// TIA Portal V19 export
FUNCTION "MeasWheelCheckRotation_TypeExtEnc" : Int   // FC49, LAD
TITLE = Check velocity of the measuring wheel compared with velocity axis (motor)
// Da usare con encoder rotella di misura collegata come encoder esterno e che quindi non chiude l'anello di posizione di un asse
// stored: Access Published, SetENOAutomatically false
   VAR_INPUT
      TO_EncMatCounter : TO_ExternalEncoder;   // TO of the external encoder
      VelMaterialMover : LReal;   // "#TO_Ax.Velocity"of the material mover axis
      VelMin : LReal;   // Min velocity for execute check
      ErrPercentageMax : LReal;   // Max error % beetween velocity
   END_VAR
   VAR_OUTPUT
      Err : LReal;   // Show % actual error percentage
   END_VAR
   VAR_TEMP
      MeasWheelIsActive : Bool;
      MotorVelocity : LReal;
      MotorVelocityABS : LReal;
      ErrorPercentage : LReal;
      Check : Bool;
      err0 : LReal;
   END_VAR
   VAR CONSTANT
      RET_NULL : Int := 0;
      RET_VEL_OK : Int := 1;
      RET_VEL_BELOW_MIN : Int := 10;
      RET_ERR_ENC_NOT_VALID : Int := 101;
      RET_VEL_DELTA_EXCEED : Int := 103;
   END_VAR
   VAR_TEMP   // added for the SCL form of the ladder/FBD networks
      _w1 : Bool;
   END_VAR
BEGIN

REGION Network 1: Out error percentage
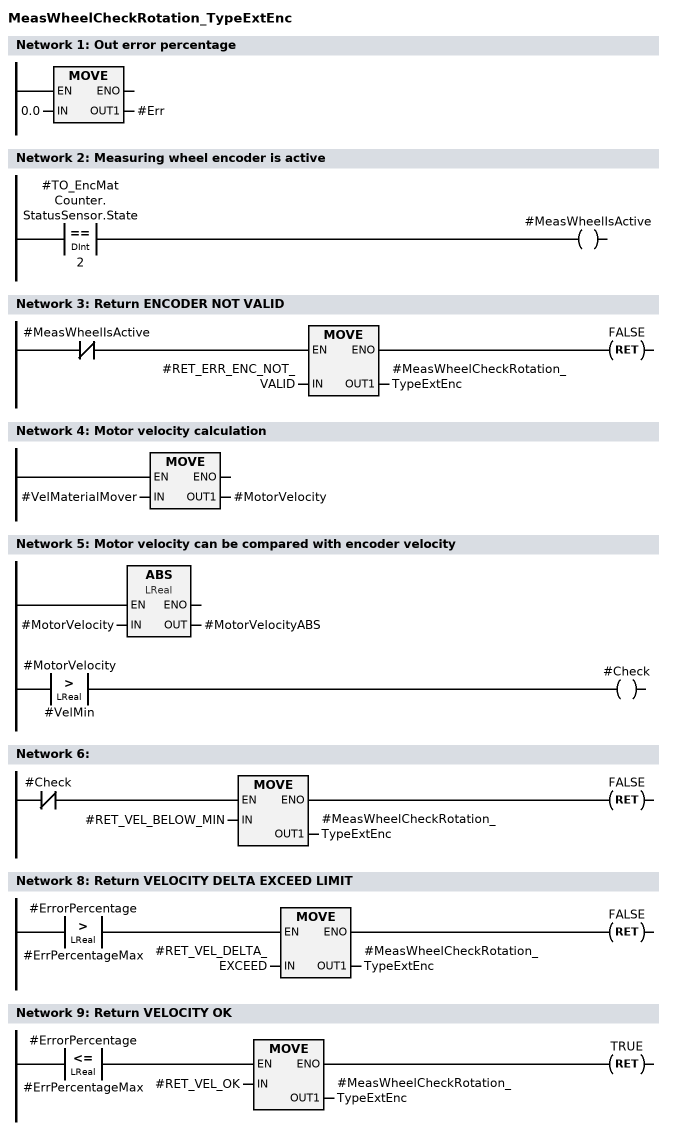
   RUNG wire#powerrail
      { S7_GenerateENO := "TRUE" } Move(in := 0.0, out1 => #Err)
   END_RUNG
   // the same network as SCL:
   #Err := 0.0;
END_REGION

REGION Network 2: Measuring wheel encoder is active
   RUNG wire#powerrail
      { S7_Templates := "SrcType := DInt" } EQ_Contact(in1 := #TO_EncMatCounter.StatusSensor.State, in2 := 2)
      Coil( #MeasWheelIsActive )
   END_RUNG
   // the same network as SCL:
   #MeasWheelIsActive := #TO_EncMatCounter.StatusSensor.State = 2;
END_REGION

REGION Network 3: Return ENCODER NOT VALID
   RUNG wire#powerrail
      I_Contact( #MeasWheelIsActive )
      { S7_GenerateENO := "TRUE" } Move(in := #RET_ERR_ENC_NOT_VALID, out1 => #MeasWheelCheckRotation_TypeExtEnc)
      ReturnCoil( FALSE )
   END_RUNG
   // the same network as SCL:
   // ENO of a box is taken as its EN; it also drops when the box reports an error
   IF NOT #MeasWheelIsActive THEN
       #MeasWheelCheckRotation_TypeExtEnc := #RET_ERR_ENC_NOT_VALID;
       ENO := FALSE;
       RETURN;
   END_IF;
END_REGION

REGION Network 4: Motor velocity calculation
   RUNG wire#powerrail
      { S7_GenerateENO := "TRUE" } Move(in := #VelMaterialMover, out1 => #MotorVelocity)
   END_RUNG
   // the same network as SCL:
   #MotorVelocity := #VelMaterialMover;
END_REGION

REGION Network 5: Motor velocity can be compared with encoder velocity
   RUNG wire#powerrail
      { S7_Templates := "SrcType := LReal"; S7_GenerateENO := "TRUE" } Abs(in := #MotorVelocity, out => #MotorVelocityABS)
   END_RUNG
   RUNG wire#powerrail
      { S7_Templates := "SrcType := LReal" } GT_Contact(in1 := #MotorVelocity, in2 := #VelMin)
      Coil( #Check )
   END_RUNG
   // the same network as SCL:
   #MotorVelocityABS := ABS(#MotorVelocity);
   #Check := #MotorVelocity > #VelMin;
END_REGION

REGION Network 6
   RUNG wire#powerrail
      I_Contact( #Check )
      { S7_GenerateENO := "TRUE" } Move(in := #RET_VEL_BELOW_MIN, out1 => #MeasWheelCheckRotation_TypeExtEnc)
      ReturnCoil( FALSE )
   END_RUNG
   // the same network as SCL:
   // ENO of a box is taken as its EN; it also drops when the box reports an error
   IF NOT #Check THEN
       #MeasWheelCheckRotation_TypeExtEnc := #RET_VEL_BELOW_MIN;
       ENO := FALSE;
       RETURN;
   END_IF;
END_REGION

REGION Network 7 (SCL): Error percentage between motor and encoder

   #err0 := ABS(#TO_EncMatCounter.StatusExtrapolation.ExtrapolatedVelocity - #MotorVelocity);

   #ErrorPercentage := 100.0 * #err0 / #TO_EncMatCounter.StatusExtrapolation.ExtrapolatedVelocity;


   #Err := #ErrorPercentage;
END_REGION

REGION Network 8: Return VELOCITY DELTA EXCEED LIMIT
   RUNG wire#powerrail
      { S7_Templates := "SrcType := LReal" } GT_Contact(in1 := #ErrorPercentage, in2 := #ErrPercentageMax)
      { S7_GenerateENO := "TRUE" } Move(in := #RET_VEL_DELTA_EXCEED, out1 => #MeasWheelCheckRotation_TypeExtEnc)
      ReturnCoil( FALSE )
   END_RUNG
   // the same network as SCL:
   // ENO of a box is taken as its EN; it also drops when the box reports an error
   #_w1 := #ErrorPercentage > #ErrPercentageMax;
   IF #_w1 THEN
       #MeasWheelCheckRotation_TypeExtEnc := #RET_VEL_DELTA_EXCEED;
       ENO := FALSE;
       RETURN;
   END_IF;
END_REGION

REGION Network 9: Return VELOCITY OK
   RUNG wire#powerrail
      { S7_Templates := "SrcType := LReal" } LE_Contact(in1 := #ErrorPercentage, in2 := #ErrPercentageMax)
      { S7_GenerateENO := "TRUE" } Move(in := #RET_VEL_OK, out1 => #MeasWheelCheckRotation_TypeExtEnc)
      ReturnCoil( TRUE )
   END_RUNG
   // the same network as SCL:
   // ENO of a box is taken as its EN; it also drops when the box reports an error
   #_w1 := #ErrorPercentage <= #ErrPercentageMax;
   IF #_w1 THEN
       #MeasWheelCheckRotation_TypeExtEnc := #RET_VEL_OK;
       ENO := TRUE;
       RETURN;
   END_IF;
END_REGION
END_FUNCTION
